INTERFACE IDisposable EXTENDS __System.IQueryInterface

METHOD Dispose
END_METHOD

END_INTERFACE

(* stored: Version 1.1.0.1
   Itf IDisposable: Id {741731d5-d4c2-417d-b103-36d0222459a8}
   Method Dispose: Id {34c9bfbf-6577-4284-bd10-d202ab5bd94a} *)
